{attribute 'qualified_only'}
{attribute 'strict'}
{attribute 'to_string'}
TYPE EAnlagenStatus:
(
	OFF := 0,
	StateInitOpen := 10,
	StateInitClose := 11,
	StateReady := 20,
	StateProductionOpen := 30,
	StateProductionClose := 31,
	StateDone := 40	
);
END_TYPE

(* stored: Version 1.1.0.1
   DUT EAnlagenStatus: Id {519a8894-b0e0-430f-8d08-ab5e09460af9} *)
